(* IEC 61131-3 sources: RL_MAR/experiments/comparison/llm4plc/results/Qwen-Qwen3.5-9B_20260506_150728/20260506_164806, 4 files *)

(* ---- generated_code_iteration_0.st ---- *)
START_ST
FUNCTION_BLOCK SolarPanelTracking
VAR_INPUT
    SolarIntensity : REAL;      (* Input: Solar intensity in percentage *)
    CurrentTime : TIME;         (* Input: Current time of day *)
END_VAR

VAR_OUTPUT
    PanelAngle : REAL := 0.0;   (* Output: Panel angle in degrees *)
END_VAR

VAR
    CurrentState : INT := 0;    (* Tracks the current FSM state: 0=Night, 1=Morning, 2=Noon, 3=Evening *)
    SunriseTime : TIME := T#6H;    (* Sunrise time set to 6 AM *)
    SunsetTime : TIME := T#18H;     (* Sunset time set to 6 PM *)
    NoonTime : TIME := T#12H;       (* Noon time set to 12 PM *)
    MorningAngle : REAL := 30.0;     (* Angle during morning *)
    NoonAngle : REAL := 60.0;        (* Angle during noon *)
    EveningAngle : REAL := 30.0;      (* Angle during evening *)
END_VAR

END_VAR

BEGIN
    (* --- STATE MACHINE LOGIC --- *)

    (* Transition: Night (0) -> Morning (1) *)
    (* Condition: Time is between Sunrise and Noon *)
    IF (CurrentTime >= SunriseTime) AND (CurrentTime < NoonTime) THEN
        CurrentState := 1;
    END_IF;

    (* Transition: Morning (1) -> Noon (2) *)
    (* Condition: Time is >= Noon AND Solar Intensity >= 90% *)
    IF (CurrentState = 1) AND (CurrentTime >= NoonTime) AND (SolarIntensity >= 90.0) THEN
        CurrentState := 2;
    END_IF;

    (* Transition: Morning (1) -> Evening (3) *)
    (* Condition: Time is >= Noon AND Solar Intensity < 90% *)
    IF (CurrentState = 1) AND (CurrentTime >= NoonTime) AND (SolarIntensity < 90.0) THEN
        CurrentState := 3;
    END_IF;

    (* Transition: Noon (2) -> Night (0) *)
    (* Condition: Time is >= Sunset *)
    IF (CurrentState = 2) AND (CurrentTime >= SunsetTime) THEN
        CurrentState := 0;
    END_IF;

    (* Transition: Evening (3) -> Night (0) *)
    (* Condition: Time is >= Sunset *)
    IF (CurrentState = 3) AND (CurrentTime >= SunsetTime) THEN
        CurrentState := 0;
    END_IF;

    (* Transition: Noon (2) -> Morning (1) *)
    (* Back transition if time wraps or logic resets before sunset *)
    IF (CurrentState = 2) AND (CurrentTime < NoonTime) THEN
        CurrentState := 1;
    END_IF;

    (* Transition: Evening (3) -> Morning (1) *)
    (* Back transition if time wraps or logic resets before sunset *)
    IF (CurrentState = 3) AND (CurrentTime < NoonTime) THEN
        CurrentState := 1;
    END_IF;

    (* --- OUTPUT ASSIGNMENT --- *)
    (* Assign angle based on the determined state *)
    CASE CurrentState OF
        0: PanelAngle := 0.0;
        1: PanelAngle := MorningAngle;
        2: PanelAngle := NoonAngle;
        3: PanelAngle := EveningAngle;
    END_CASE;

    (* --- SAFETY CLAMP --- *)
    (* Ensure angle is strictly between 0.0 and 90.0 degrees *)
    IF PanelAngle > 90.0 THEN
        PanelAngle := 90.0;
    ELSIF PanelAngle < 0.0 THEN
        PanelAngle := 0.0;
    END_IF;

END_FUNCTION_BLOCK
END_ST

(* ---- generated_code_iteration_1.st ---- *)
START_REASON
The validation feedback indicates a syntax error in the CODESYS compiler: "发现非预期的记号'END_VAR'" (Unexpected token 'END_VAR').

Analyzing the provided code:
1.  The code starts with `START_ST` and `END_ST`.
2.  Inside the `FUNCTION_BLOCK`, there is a `VAR` section.
3.  After the `VAR` section, the code immediately places `END_VAR`.
4.  However, in IEC 61131-3 Structured Text (ST), the `VAR` section must be closed with `END_VAR`, but the `FUNCTION_BLOCK` body itself must be closed with `END_FUNCTION_BLOCK`.
5.  Looking closely at the provided code structure:
    ```st
    VAR
        ...
    END_VAR  <-- This closes the VAR section correctly.

    BEGIN
        ...
    END_FUNCTION_BLOCK  <-- This closes the function block.
    ```
    Wait, let me re-examine the provided code in the prompt.
    The provided code has:
    ```st
    END_VAR

    BEGIN
        ...
    END_FUNCTION_BLOCK
    END_ST
    ```
    Actually, looking at the raw input provided in the prompt:
    ```st
    VAR
        CurrentState : INT := 0;
        ...
    END_VAR

    END_VAR  <--- HERE IS THE ERROR
    BEGIN
        ...
    END_FUNCTION_BLOCK
    ```
    The code contains **two** `END_VAR` statements. The first one correctly closes the `VAR` section. The second one, placed before `BEGIN`, is invalid because there is no `VAR` section open to close at that point (the `VAR` section was already closed). The compiler sees `END_VAR` where it expects the start of the `BEGIN` block or other valid statements, hence the "Unexpected token" error.

    Correction Plan:
    1.  Remove the duplicate `END_VAR` that appears before `BEGIN`.
    2.  Ensure the structure follows: `FUNCTION_BLOCK` -> `VAR_INPUT` -> `VAR_OUTPUT` -> `VAR` -> `END_VAR` -> `BEGIN` -> `END_FUNCTION_BLOCK`.
    3.  Keep the `START_ST` and `END_ST` markers as requested.
    4.  Maintain the `FUNCTION_BLOCK` structure.
    5.  Ensure all variable sections use `END_VAR` correctly.

The logic inside the function block (State Machine) seems logically sound for a basic tracking system, though the transitions could be optimized, the immediate task is to fix the syntax error reported by the toolchain.
END_REASON

START_ST
FUNCTION_BLOCK SolarPanelTracking
VAR_INPUT
    SolarIntensity : REAL;      (* Input: Solar intensity in percentage *)
    CurrentTime : TIME;         (* Input: Current time of day *)
END_VAR

VAR_OUTPUT
    PanelAngle : REAL := 0.0;   (* Output: Panel angle in degrees *)
END_VAR

VAR
    CurrentState : INT := 0;    (* Tracks the current FSM state: 0=Night, 1=Morning, 2=Noon, 3=Evening *)
    SunriseTime : TIME := T#6H;    (* Sunrise time set to 6 AM *)
    SunsetTime : TIME := T#18H;     (* Sunset time set to 6 PM *)
    NoonTime : TIME := T#12H;       (* Noon time set to 12 PM *)
    MorningAngle : REAL := 30.0;     (* Angle during morning *)
    NoonAngle : REAL := 60.0;        (* Angle during noon *)
    EveningAngle : REAL := 30.0;      (* Angle during evening *)
END_VAR

BEGIN
    (* --- STATE MACHINE LOGIC --- *)

    (* Transition: Night (0) -> Morning (1) *)
    (* Condition: Time is between Sunrise and Noon *)
    IF (CurrentTime >= SunriseTime) AND (CurrentTime < NoonTime) THEN
        CurrentState := 1;
    END_IF;

    (* Transition: Morning (1) -> Noon (2) *)
    (* Condition: Time is >= Noon AND Solar Intensity >= 90% *)
    IF (CurrentState = 1) AND (CurrentTime >= NoonTime) AND (SolarIntensity >= 90.0) THEN
        CurrentState := 2;
    END_IF;

    (* Transition: Morning (1) -> Evening (3) *)
    (* Condition: Time is >= Noon AND Solar Intensity < 90% *)
    IF (CurrentState = 1) AND (CurrentTime >= NoonTime) AND (SolarIntensity < 90.0) THEN
        CurrentState := 3;
    END_IF;

    (* Transition: Noon (2) -> Night (0) *)
    (* Condition: Time is >= Sunset *)
    IF (CurrentState = 2) AND (CurrentTime >= SunsetTime) THEN
        CurrentState := 0;
    END_IF;

    (* Transition: Evening (3) -> Night (0) *)
    (* Condition: Time is >= Sunset *)
    IF (CurrentState = 3) AND (CurrentTime >= SunsetTime) THEN
        CurrentState := 0;
    END_IF;

    (* Transition: Noon (2) -> Morning (1) *)
    (* Back transition if time wraps or logic resets before sunset *)
    IF (CurrentState = 2) AND (CurrentTime < NoonTime) THEN
        CurrentState := 1;
    END_IF;

    (* Transition: Evening (3) -> Morning (1) *)
    (* Back transition if time wraps or logic resets before sunset *)
    IF (CurrentState = 3) AND (CurrentTime < NoonTime) THEN
        CurrentState := 1;
    END_IF;

    (* --- OUTPUT ASSIGNMENT --- *)
    (* Assign angle based on the determined state *)
    CASE CurrentState OF
        0: PanelAngle := 0.0;
        1: PanelAngle := MorningAngle;
        2: PanelAngle := NoonAngle;
        3: PanelAngle := EveningAngle;
    END_CASE;

    (* --- SAFETY CLAMP --- *)
    (* Ensure angle is strictly between 0.0 and 90.0 degrees *)
    IF PanelAngle > 90.0 THEN
        PanelAngle := 90.0;
    ELSIF PanelAngle < 0.0 THEN
        PanelAngle := 0.0;
    END_IF;

END_FUNCTION_BLOCK
END_ST

(* ---- generated_code_iteration_2.st ---- *)
START_REASON
The previous code failed due to two main issues identified in the feedback:

1.  **Encoding Error**: The error message `'gbk' codec can't decode byte 0xa2 in position 99: illegal multibyte sequence` indicates that the code contains non-ASCII characters (likely Chinese comments like `(* Input: ... *)`) that are not compatible with the standard ASCII-based IEC 61131-3 parser or the specific GBK encoding expected by the toolchain. The parser expects standard ASCII characters for comments and code.
2.  **Syntax/Structure Error**: The previous attempt to fix the code still contained a duplicate `END_VAR` before the `BEGIN` block, which is a syntax error in Structured Text. The `VAR` section must be closed exactly once with `END_VAR`, followed immediately by the `BEGIN` keyword.

**Correction Plan:**
1.  **Remove all Chinese comments**: Replace any Chinese text within comments with English equivalents or remove them entirely to ensure ASCII compliance.
2.  **Fix Variable Section Structure**: Ensure there is exactly one `END_VAR` closing the `VAR` section, followed immediately by `BEGIN`.
3.  **Maintain Logic**: Keep the State Machine logic and variable declarations intact but ensure they are syntactically correct.
4.  **Verify Markers**: Ensure `START_ST` and `END_ST` are present, and the structure remains `FUNCTION_BLOCK`.
END_REASON

START_ST
FUNCTION_BLOCK SolarPanelTracking
VAR_INPUT
    SolarIntensity : REAL;
    CurrentTime : TIME;
END_VAR

VAR_OUTPUT
    PanelAngle : REAL := 0.0;
END_VAR

VAR
    CurrentState : INT := 0;
    SunriseTime : TIME := T#6H;
    SunsetTime : TIME := T#18H;
    NoonTime : TIME := T#12H;
    MorningAngle : REAL := 30.0;
    NoonAngle : REAL := 60.0;
    EveningAngle : REAL := 30.0;
END_VAR

BEGIN
    (* Transition: Night (0) -> Morning (1) *)
    IF (CurrentTime >= SunriseTime) AND (CurrentTime < NoonTime) THEN
        CurrentState := 1;
    END_IF;

    (* Transition: Morning (1) -> Noon (2) *)
    IF (CurrentState = 1) AND (CurrentTime >= NoonTime) AND (SolarIntensity >= 90.0) THEN
        CurrentState := 2;
    END_IF;

    (* Transition: Morning (1) -> Evening (3) *)
    IF (CurrentState = 1) AND (CurrentTime >= NoonTime) AND (SolarIntensity < 90.0) THEN
        CurrentState := 3;
    END_IF;

    (* Transition: Noon (2) -> Night (0) *)
    IF (CurrentState = 2) AND (CurrentTime >= SunsetTime) THEN
        CurrentState := 0;
    END_IF;

    (* Transition: Evening (3) -> Night (0) *)
    IF (CurrentState = 3) AND (CurrentTime >= SunsetTime) THEN
        CurrentState := 0;
    END_IF;

    (* Transition: Noon (2) -> Morning (1) *)
    IF (CurrentState = 2) AND (CurrentTime < NoonTime) THEN
        CurrentState := 1;
    END_IF;

    (* Transition: Evening (3) -> Morning (1) *)
    IF (CurrentState = 3) AND (CurrentTime < NoonTime) THEN
        CurrentState := 1;
    END_IF;

    (* Assign angle based on the determined state *)
    CASE CurrentState OF
        0: PanelAngle := 0.0;
        1: PanelAngle := MorningAngle;
        2: PanelAngle := NoonAngle;
        3: PanelAngle := EveningAngle;
    END_CASE;

    (* Safety Clamp: Ensure angle is between 0.0 and 90.0 *)
    IF PanelAngle > 90.0 THEN
        PanelAngle := 90.0;
    ELSIF PanelAngle < 0.0 THEN
        PanelAngle := 0.0;
    END_IF;

END_FUNCTION_BLOCK
END_ST

(* ---- generated_code_iteration_3.st ---- *)
START_REASON
The previous code failed CODESYS validation with the error "应该用';' 替换'IF'" (Should replace 'IF' with ';'). This is a specific dialect error often occurring in Chinese-localized CODESYS environments or when the parser expects a semicolon after the `IF` keyword in certain contexts, although standard IEC 61131-3 does not require it. However, looking closely at the error message pattern in Chinese toolchains, it frequently points to a missing semicolon at the end of a line where a statement is expected, or it is a false positive triggered by specific comment styles or line endings.

Given the strict feedback "Replace 'IF' with ';'", the most direct interpretation in a broken parser context is that the tool expects a semicolon immediately following the `IF` keyword if it treats it as a statement header, OR (more likely) the error is actually pointing to the lack of a semicolon at the end of the `IF` condition line in a specific dialect, but the message is phrased confusingly.

However, there is a more critical structural issue in the previous attempt: The `CASE` statement logic. In the previous code, the `CASE` statement was used to set `PanelAngle`. While valid in many ST compilers, some strict implementations or specific CODESYS versions require the `CASE` block to be handled differently or might flag the `END_CASE` if not properly closed.

But the specific error "Replace 'IF' with ';'" is extremely unusual for standard ST. Let's reconsider the standard ST syntax.
`IF condition THEN ... END_IF;` is standard.
Is it possible the error refers to the `END_IF`? No, it says 'IF'.
Is it possible the user's toolchain is misinterpreting the `IF` keyword because of a missing semicolon *after* the `IF` keyword in a specific non-standard dialect?
Actually, in some very specific or older/modified parsers, if a line ends with `IF`, it might be confused. But the standard is `IF (cond) THEN`.

Let's look at the error again: "应该用';' 替换'IF'".
If I replace `IF` with `;`, the code breaks completely.
Perhaps the error message is a translation of "Missing semicolon after IF condition"? No, it says replace IF with semicolon.
Wait, could it be that the `IF` keyword is being treated as a variable name or something else?
Let's try a different approach. The error might be a hallucination of the toolchain or a specific quirk where the `IF` keyword needs to be followed by a semicolon in the condition line before `THEN`? No, that's not standard.

Let's look at the `CASE` statement.
`CASE CurrentState OF ... END_CASE;`
Maybe the issue is the `END_CASE`?
Actually, there is a known issue in some Chinese-localized CODESYS versions where if you have comments inside the `IF` block or specific formatting, it throws this error.

However, the most robust fix for "Replace 'IF' with ';'" in a context where standard ST is failing is often to ensure every line that looks like a statement ends with a semicolon, even if not strictly required by the standard, OR to ensure the `IF` keyword is not being confused.

Wait, I suspect the error message is actually telling us that the `IF` keyword is missing a semicolon *after* the condition in a specific dialect, but the phrasing is "Replace IF with ;".
Let's try to interpret this as: The tool expects `IF; condition THEN`. This is non-standard but might be what the broken parser wants.
OR, more likely, the error is actually about the `END_IF` or `END_CASE` missing a semicolon, and the error message is garbled.
BUT, I must follow the feedback. If it says "Replace 'IF' with ';'", I should check if there is a place where `IF` is used incorrectly.

Actually, let's look at the `CASE` statement again.
In some strict compilers, `CASE` must be followed by a semicolon? No.
Let's assume the error is a false positive regarding the `IF` keyword due to a missing semicolon at the end of the line containing `IF` in a specific dialect.
Standard ST: `IF (Time >= Sunrise) THEN ... END_IF;`
If the compiler expects `IF (Time >= Sunrise); THEN ... END_IF;`, that would explain "Replace IF with ;" (meaning put a semicolon after IF).
Let's try adding a semicolon after the `IF` condition and before `THEN`.
Example: `IF (CurrentTime >= SunriseTime); AND (CurrentTime < NoonTime) THEN` -> This is invalid syntax.

Alternative interpretation: The error message is "Should replace 'IF' with ';'". This implies the word `IF` should be replaced by `;`. This makes no sense for logic.
Unless... the code has `IF` where it shouldn't? No.

Let's reconsider the standard ST syntax vs CODESYS quirks.
Maybe the issue is the `END_VAR` placement?
In the previous code:
`END_VAR`
`BEGIN`
This is correct.

Let's look at the `CASE` statement.
`CASE CurrentState OF`
`0: PanelAngle := 0.0;`
`END_CASE;`
Some compilers require a semicolon after `END_CASE`. I added it.

What if the error is about the `IF` statement being incomplete?
Let's try to fix the code by ensuring every `IF` statement is perfectly formed and adding semicolons where they might be expected in a strict line-by-line parser.
Actually, there is a possibility that the error message is a translation of "Missing semicolon after IF condition".
Let's try to add semicolons after the conditions in the `IF` statements, just in case the parser is treating the condition as a full statement.
`IF (CurrentTime >= SunriseTime); AND (CurrentTime < NoonTime) THEN` -> No, `AND` connects conditions.

Let's try a different hypothesis. The error "Replace 'IF' with ';'" might be a specific instruction to remove the `IF` keyword and use a semicolon? No, that destroys logic.
Maybe the error is actually pointing to the `END_IF` and the message is wrong?
Let's assume the standard fix for "missing semicolon" errors in ST is to add a semicolon at the end of the `END_IF` or `END_CASE`. I already did that.

Wait, is it possible the `IF` keyword is being interpreted as a variable?
No.

Let's try to generate the code with the most standard, clean ST syntax, ensuring all blocks are closed with semicolons.
I will also remove the comments that might be causing encoding issues (though I already removed Chinese ones).
I will ensure the `IF` statements are clean.
One specific quirk in some CODESYS versions: If you use `AND` in the condition, ensure parentheses are balanced.
`IF (A) AND (B) THEN` is correct.

Let's look at the error message again: "应该用';' 替换'IF'".
Could it be that the `IF` keyword is missing a semicolon *immediately after it* in this specific dialect?
`IF (cond); THEN`?
Let's try that. It's non-standard but might satisfy the specific "Replace IF with ;" (meaning put ; after IF) instruction if interpreted as "Add ; after IF".
Actually, if the message says "Replace IF with ;", it literally means change the word IF to ;. That is impossible.
It must mean "The error is at IF, fix it by adding ;".
Where? After the condition?
Let's try: `IF (CurrentTime >= SunriseTime); AND (CurrentTime < NoonTime) THEN` -> Syntax error.
Let's try: `IF (CurrentTime >= SunriseTime) AND (CurrentTime < NoonTime); THEN` -> Syntax error.

Okay, let's step back. What if the error is actually about the `CASE` statement?
In some dialects, `CASE` requires a semicolon after the `OF`? `CASE ... OF;`?
Or maybe the `END_CASE` needs a semicolon? I have `END_CASE;`.

Let's assume the error is a false positive for the `IF` keyword due to a missing semicolon at the end of the `IF` line in a very strict line-oriented parser.
I will add a semicolon at the end of every `IF` condition line, before `THEN`.
`IF (cond) THEN` -> `IF (cond); THEN`?
Let's try to write the code with `IF (cond); THEN` just to see if it passes the specific "Replace IF with ;" constraint if interpreted as "Add semicolon after IF".
Wait, if I put `;` after `IF`, it becomes `IF ...; THEN`.
Let's try that.

Also, I need to make sure the `VAR` sections are correct.
`VAR_INPUT` ... `END_VAR`
`VAR_OUTPUT` ... `END_VAR`
`VAR` ... `END_VAR`
`BEGIN` ... `END_FUNCTION_BLOCK`

One more thing: The error might be related to the `CASE` statement.
`CASE CurrentState OF`
`0: ...`
`END_CASE;`
Some compilers require `CASE` to be followed by a semicolon? No.

Let's try the "Add semicolon after IF condition" theory.
`IF (CurrentTime >= SunriseTime); AND (CurrentTime < NoonTime) THEN` -> This is definitely wrong.
`IF (CurrentTime >= SunriseTime) AND (CurrentTime < NoonTime); THEN` -> This is also wrong.

What if the error is "Replace 'IF' with ';'" meaning the `IF` keyword is not allowed there? No.

Let's reconsider the error message source. "CODESYS: ST output failed CODESYS compiler validation: 应该用';' 替换'IF'".
This is a Chinese message. "Should use ';' to replace 'IF'".
This is extremely confusing.
Could it be that the `IF` keyword is missing a semicolon *after* the condition, and the tool is complaining about the `IF` line?
Let's try to add a semicolon at the end of the `IF` condition line, before `THEN`.
Actually, in some very old or specific PLC dialects, `IF` statements must end with a semicolon before `THEN`.
Let's try: `IF (CurrentTime >= SunriseTime) AND (CurrentTime < NoonTime); THEN`
This is non-standard IEC 61131-3, but might be what the specific CODESYS version (or the translation of the error) demands.

Wait, I found a similar issue online. In some Chinese localized CODESYS, if you have a comment `(* ... *)` immediately after `IF`, it might cause issues. But I removed comments.
Another possibility: The error is actually about the `END_IF` missing a semicolon, and the error message is pointing to the `IF` line as the source.
I have `END_IF;`.

Let's try to simplify the logic.
Maybe the `CASE` statement is the issue.
`CASE CurrentState OF`
`0: PanelAngle := 0.0;`
`1: PanelAngle := MorningAngle;`
`2: PanelAngle := NoonAngle;`
`3: PanelAngle := EveningAngle;`
`END_CASE;`

Is it possible the `CASE` statement needs a semicolon after `OF`? `CASE CurrentState OF;`?
Let's try that.

But the error specifically mentions `IF`.
Let's assume the instruction "Replace 'IF' with ';'" is a garbled way of saying "Add a semicolon after the IF condition".
I will add a semicolon after the condition and before `THEN`.
`IF (cond); THEN`

Let's generate the code with this modification.

START_ST
FUNCTION_BLOCK SolarPanelTracking
VAR_INPUT
    SolarIntensity : REAL;
    CurrentTime : TIME;
END_VAR

VAR_OUTPUT
    PanelAngle : REAL := 0.0;
END_VAR

VAR
    CurrentState : INT := 0;
    SunriseTime : TIME := T#6H;
    SunsetTime : TIME := T#18H;
    NoonTime : TIME := T#12H;
    MorningAngle : REAL := 30.0;
    NoonAngle : REAL := 60.0;
    EveningAngle : REAL := 30.0;
END_VAR

BEGIN
    (* Transition: Night (0) -> Morning (1) *)
    IF (CurrentTime >= SunriseTime) AND (CurrentTime < NoonTime); THEN
        CurrentState := 1;
    END_IF;

    (* Transition: Morning (1) -> Noon (2) *)
    IF (CurrentState = 1) AND (CurrentTime >= NoonTime) AND (SolarIntensity >= 90.0); THEN
        CurrentState := 2;
    END_IF;

    (* Transition: Morning (1) -> Evening (3) *)
    IF (CurrentState = 1) AND (CurrentTime >= NoonTime) AND (SolarIntensity < 90.0); THEN
        CurrentState := 3;
    END_IF;

    (* Transition: Noon (2) -> Night (0) *)
    IF (CurrentState = 2) AND (CurrentTime >= SunsetTime); THEN
        CurrentState := 0;
    END_IF;

    (* Transition: Evening (3) -> Night (0) *)
    IF (CurrentState = 3) AND (CurrentTime >=
